Yaskawa INFORM job: TEST_ID.JBI

/JOB
//NAME TEST_ID
///FOLDERNAME TEST_JOBS
//POS
///NPOS 0,0,0,0,0,0
//INST
///DATE 2023/05/03 16:52
///COMM TEST ID SETTINGS
///ATTR SC,RW
///GROUP1 RB1
NOP
CALL JOB:TRIGGER_RESET
'--------------------------------
'IDs Eingeben
CALL JOB:SET_ID ARGF0 ARGF"WID"
CALL JOB:SET_ID ARGF3 ARGF"NAHT_NR"
CALL JOB:SET_ID ARGF2 ARGF"LAGE_NR"
CALL JOB:SET_ID ARGF4 ARGF"RAUPE_NR"
CALL JOB:SET_ID ARGF5 ARGF"SCHW_NR"
'--------------------------------
'Scope Aufnahme starten
CALL JOB:TRIGGER ARGF"PROGRAMM_EIN"
'--------------------------------
'IDs ändern
TIMER T=2.00
CALL JOB:INC_NR ARGF"SCHW_NR"
TIMER T=2.00
CALL JOB:INC_NR ARGF"RAUPE_NR"
TIMER T=2.00
CALL JOB:INC_NR ARGF"LAGE_NR"
TIMER T=2.00
CALL JOB:INC_NR ARGF"SCHW_NR"
TIMER T=2.00
CALL JOB:INC_NR ARGF"LAGE_NR"
TIMER T=2.00
CALL JOB:TRIGGER ARGF"SCHWEISSEN_EIN"
TIMER T=1.00
CALL JOB:TRIGGER ARGF"SCHWEISSEN_AUS"
TIMER T=1.00
CALL JOB:TRIGGER ARGF"SCHWEISSEN_EIN"
TIMER T=1.00
CALL JOB:TRIGGER ARGF"SCHWEISSEN_AUS"
TIMER T=1.00
CALL JOB:TRIGGER ARGF"SCHWEISSEN_EIN"
TIMER T=1.00
CALL JOB:TRIGGER ARGF"SCHWEISSEN_AUS"
TIMER T=1.00
CALL JOB:INC_NR ARGF"NAHT_NR"
TIMER T=2.00
'--------------------------------
'Nummern direkt setzen
CALL JOB:SET_IDS ARGF2 ARGF3 ARGF4 ARGF5
TIMER T=2.00
'--------------------------------
'IDs direkt setzen
CALL JOB:SET_IDS_FULL ARGF10 ARGF20 ARGF30 ARGF40 ARGF50
TIMER T=2.00
'--------------------------------
'Scope Aufnahme stoppen
CALL JOB:TRIGGER ARGF"PROGRAMM_AUS"
'--------------------------------
'CLEANUP
CALL JOB:TRIGGER_RESET
END
